INTERFACE I_Focus

METHOD SetFocus : BOOL
VAR_INPUT
	Focus	: LREAL;
END_VAR
END_METHOD

END_INTERFACE

(* stored: Version 1.1.0.1, ProductVersion 3.1.4024.13
   POU I_Focus: Id {caac64bd-2b24-42ed-9fda-2fff76bfb76e}, SpecialFunc None
   Method SetFocus: Id {8b7d991c-9a45-4faf-a402-2c683bc45831} *)
